PROGRAM Alarm_System
VAR
	bIsInitialized : BOOL;
	bEmergency : BOOL;
END_VAR

IF NOT bIsInitialized THEN	// Initialization, since functions can't run in top pane
	bIsInitialized := TRUE;
	gAL.fbAlarm.CreateEx(TC_Events.TankAlarmEvent.Emergency, TRUE, 0);
END_IF

IF bEmergency THEN
	bEmergency := FALSE;
	gAL.fbAlarm.Raise(0); // 0 -> Current time
END_IF

// NOT USED AT THE MOMENT OH MA GAH !

END_PROGRAM

(* stored: Version 1.1.0.1, ProductVersion 3.1.4024.12
   POU Alarm_System: Id {0c25327a-9784-407a-9f83-71ce43145858}, SpecialFunc None *)
